// TIA Portal project "ContactorControlObject_HmiVideo_v2" (V16)

(* hardware
DEVICE "ET 200SP station_1"  ET 200SP-Station
   slot 0: "Rack_0"  Rack  6ES5 710-8MAx1
   slot 1: "PLC_1"  CPU 1510SP-1 PN  6ES7 510-1DJ00-0AB0  V1.8
      slot 32768: "PROFINET interface_1"  X1
         slot 32771: "Port_3"  X1 P3
   slot 2: "Server module_1"  Server module  6ES7 193-6PA00-0AA0  V1.1
      slot 1: "Server module_1"  Server module
   slot 127: "BA 2xRJ45"  BA 2xRJ45  6ES7 193-6AR00-0AA0  V0.0
      slot 32769: "Port_1"  X1 P1  6ES7 193-6AR00-0AA0
      slot 32770: "Port_2"  X1 P2  6ES7 193-6AR00-0AA0
DEVICE "HMI_1"  KTP400 Comfort
   slot 0: "HMI_1"  KTP400 Comfort  6AV2 124-2DC01-0AX0  16.0.0.0
   slot 1: "HMI_RT_1"  KTP400 Comfort  6AV2 124-2DC01-0AX0  16.0.0.0
   slot 5: "HMI_1.IE_CP_1"  PROFINET Interface  16.0.0.0
      slot 1: "PROFINET Interface_1"  PROFINET Interface
         slot 1: "Port_1"  Port
   slot 7: "HMI_1.MPI/DP_CP_1"  MPI/DP Interface  16.0.0.0
*)

// ===== PLC "PLC_1"  CPU 1510SP-1 PN =====

// folder: ContactorDataType

TYPE "tyContactor_Input"
   STRUCT
      bContactorStartRequest : Bool;
      bContactorFeedbackInput : Bool;
   END_STRUCT;
END_TYPE

TYPE "tyContactor_StaticData"
   STRUCT
      TContactorControllTimer : TON_TIME;
      TcontactorFeedBackControlTime : Time;
   END_STRUCT;
END_TYPE

TYPE "tyContactor_Main"
   STRUCT
      MachineMode : "tyMachineMode";
      ContactorInputs : "tyContactor_Input";
      ContactorOutputs : "tyContactor_Output_1";
      ContactorStatic : "tyContactor_StaticData";
      ContactorHmiInterface : "tyHmi_Interface";
   END_STRUCT;
END_TYPE

TYPE "tyHmi_Interface"
   STRUCT
      InputFromHmiToPLC : Struct
         HmiContactorStart : Bool;
         HmiContactorStop : Bool;
         OutputToHmiFromPLC : Struct
            MachineState : "tyMachineMode";
            ContactrorStatus : "tyContactor_Output_1";
         END_STRUCT;
         ConcactorStatusInt : Int;
         Internal : Struct
            ActivateFaceControllPlate : Bool;
         END_STRUCT;
      END_STRUCT;
   END_STRUCT;
END_TYPE

TYPE "tyMachineMode"
   STRUCT
      MachineInAuto : Bool;
      MachineInManual : Bool;
      MachineIn_Idle : Bool;
   END_STRUCT;
END_TYPE

TYPE "tyContactor_Output_1"
   STRUCT
      bActivateContactorCoil : Bool;
      bContactorFault : Bool;
      b_MotorIsRunning : Bool;
   END_STRUCT;
END_TYPE

// folder: (top level)

DATA_BLOCK "ContactorControll_Obj_DB"   // DB1
{ S7_Optimized_Access := 'TRUE' }
VERSION : 0.1
// stored: InstanceOfName ContactorControll_Obj
"ContactorControll_Obj"
BEGIN
END_DATA_BLOCK

FUNCTION_BLOCK "ContactorControll_Obj"   // FB1, SCL
{ S7_Optimized_Access := 'TRUE' }
VERSION : 0.1
   VAR
      MotorContactorControll : "tyContactor_Main";
   END_VAR
BEGIN
   //=============================================================================
   // Dmitri Raihtsaum - Copyright 2023
   // Created By: Dmitri Raihtsaum
   //-----------------------------------------------------------------------------
   // Tested with:   CPU 1510SP-1 PN
   // Engineering:   TIA Portal V16
   // Functionality: Contactor Control Object Hmi Control Project 
   // Date: 19.05.2023
   // Rev 0.1
   //=============================================================================


   //Mapping
   #MotorContactorControll.ContactorStatic.TcontactorFeedBackControlTime := t#2s;
   //Logic
   //Contactor Start signal 
   IF #MotorContactorControll.MachineMode.MachineInAuto THEN
       IF #MotorContactorControll.ContactorInputs.bContactorStartRequest THEN
           #MotorContactorControll.ContactorOutputs.bActivateContactorCoil := TRUE;
       END_IF;
       //Contactor Stop signal
       IF NOT #MotorContactorControll.ContactorInputs.bContactorStartRequest THEN
           #MotorContactorControll.ContactorOutputs.bActivateContactorCoil := FALSE;
       END_IF;
   END_IF;
   //Check Contactor Status 
   IF #MotorContactorControll.ContactorOutputs.bActivateContactorCoil AND #MotorContactorControll.ContactorInputs.bContactorFeedbackInput THEN
       #MotorContactorControll.ContactorOutputs.b_MotorIsRunning := TRUE;
   ELSE
       #MotorContactorControll.ContactorOutputs.b_MotorIsRunning := FALSE;
   END_IF;
   // Fault Signal
   IF #MotorContactorControll.ContactorOutputs.bActivateContactorCoil AND NOT #MotorContactorControll.ContactorInputs.bContactorFeedbackInput
       OR NOT #MotorContactorControll.ContactorOutputs.bActivateContactorCoil AND #MotorContactorControll.ContactorInputs.bContactorFeedbackInput
   THEN
       #MotorContactorControll.ContactorStatic.TContactorControllTimer(IN := TRUE,
                                                                       PT := #MotorContactorControll.ContactorStatic.TcontactorFeedBackControlTime);
   ELSE
       #MotorContactorControll.ContactorStatic.TContactorControllTimer(IN := FALSE,
                                                                       PT := t#0ms);END_IF;
   // Fault Flag
   IF #MotorContactorControll.ContactorStatic.TContactorControllTimer.Q THEN
       #MotorContactorControll.ContactorOutputs.bContactorFault := TRUE;
   ELSE
       #MotorContactorControll.ContactorOutputs.bContactorFault := FALSE;
   END_IF;
   // Hmi 
   #MotorContactorControll.ContactorHmiInterface.InputFromHmiToPLC.OutputToHmiFromPLC.MachineState := #MotorContactorControll.MachineMode; 
   #MotorContactorControll.ContactorHmiInterface.InputFromHmiToPLC.OutputToHmiFromPLC.ContactrorStatus := #MotorContactorControll.ContactorOutputs;
   //
   IF #MotorContactorControll.ContactorOutputs.b_MotorIsRunning THEN
       #MotorContactorControll.ContactorHmiInterface.InputFromHmiToPLC.ConcactorStatusInt := 1;
   ELSIF #MotorContactorControll.ContactorOutputs.bContactorFault THEN
       #MotorContactorControll.ContactorHmiInterface.InputFromHmiToPLC.ConcactorStatusInt := 2;
   ELSE
       #MotorContactorControll.ContactorHmiInterface.InputFromHmiToPLC.ConcactorStatusInt := 0;
   END_IF;
   // Manual Hmi Contorol
   IF #MotorContactorControll.MachineMode.MachineInManual THEN
       IF #MotorContactorControll.ContactorHmiInterface.InputFromHmiToPLC.HmiContactorStart THEN
           #MotorContactorControll.ContactorOutputs.bActivateContactorCoil := TRUE;
       END_IF;
       IF #MotorContactorControll.ContactorHmiInterface.InputFromHmiToPLC.HmiContactorStop THEN
           #MotorContactorControll.ContactorOutputs.bActivateContactorCoil := FALSE;
       END_IF;
   END_IF;

   // Wrong signal  Protection 
   IF NOT #MotorContactorControll.ContactorHmiInterface.InputFromHmiToPLC.HmiContactorStart AND NOT #MotorContactorControll.ContactorHmiInterface.InputFromHmiToPLC.HmiContactorStop THEN
       #MotorContactorControll.ContactorHmiInterface.InputFromHmiToPLC.HmiContactorStop := TRUE;
   END_IF;

   //Idle 
   IF #MotorContactorControll.MachineMode.MachineIn_Idle THEN
       #MotorContactorControll.ContactorOutputs.bActivateContactorCoil := FALSE;
   END_IF;

   //=============================================================================
   //END
   //=============================================================================
END_FUNCTION_BLOCK

ORGANIZATION_BLOCK "Main"   // OB1, LAD, ProgramCycle
TITLE = "Main Program Sweep (Cycle)"
{ S7_Optimized_Access := 'TRUE' }
VERSION : 0.1
   VAR_INPUT
      Initial_Call : Bool;   // Initial call of this OB
      Remanence : Bool;   // =True, if remanent data are available
   END_VAR
BEGIN

REGION Network 1
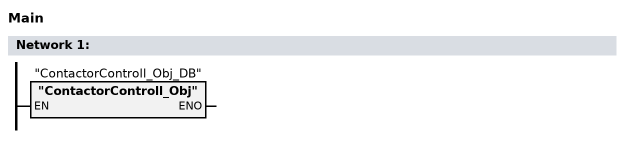
   RUNG wire#powerrail
      "ContactorControll_Obj_DB"()
   END_RUNG
   // the same network as SCL:
   "ContactorControll_Obj_DB"();   // "ContactorControll_Obj"
END_REGION
END_ORGANIZATION_BLOCK

(* ===== HMI "HMI_RT_1" =====
connection "HMI_Connection_1": ETHERNET, S7_1500_OMS

HMI tags "Fan_01"
   "Fan_01_Interface" : tyHmi_Interface = PLC ContactorControll_Obj_DB.MotorContactorControll.ContactorHmiInterface AT %DB1.DBW0, 1 s

screen "Root screen" 480x272, template "Template_1"
   ScreenModuleView "Faceplate_1_1" at 128,48 size 124x121; ScreenModuleType ""
      Guid_{11997190-9077} <- "Fan_01_Interface"
*)

(* ===== HMI "HMI_RT_1" =====

ScreenModuleEditorView "FanFacePlate" 640x480
   GraphicView "Graphic view_1" at 29,33 size 134x134; Picture "Graphic_1"
   GraphicView "Graphic view_2" at 29,33 size 134x135; Picture "Graphic_2"
   GraphicView "Graphic view_3" at 29,33 size 134x135; Picture "Graphic_3"
   Button "Button_1" at 26,31 size 139x137; TextOff 'Text'
*)

(* ===== HMI "HMI_RT_1" =====
system functions are stored by id; their names below are inferred from use

ScreenModuleEditorView "FanFacePlate" 640x480
   GraphicView "Graphic view_1" at 29,33 size 134x134; Picture "Graphic_1"
   GraphicView "Graphic view_2" at 29,33 size 134x135; Picture "Graphic_2"
      Visibility <- "Property_1.InputFromHmiToPLC.OutputToHmiFromPLC.ContactrorStatus.b_MotorIsRunning"
   GraphicView "Graphic view_3" at 29,32 size 134x135; Picture "Graphic_3"
      Visibility <- "Property_1.InputFromHmiToPLC.OutputToHmiFromPLC.ContactrorStatus.bContactorFault"
   Circle "Circle_1" at 10,10 size 173x173
      Visibility <- "Property_1.InputFromHmiToPLC.OutputToHmiFromPLC.MachineState.MachineInManual"
   Button "Button_1" at 27,32 size 139x137; TextOff 'Text'
      on Click: SetBit("Property_1.InputFromHmiToPLC.Internal.ActivateFaceControllPlate")
*)